{attribute addProperty BoxType "EL3692-0000-0017"}
{attribute addProperty Id "StatusAT %I*Status_888D5AFE1621ValueAT %I*DINT32417"}
{attribute addProperty CRC "1692878231"}
{attribute addProperty SizeInBites "48"}
{attribute addProperty SizeInBytes "6"}
TYPE SAI_Inputs_Channel_64E74597 :
STRUCT
	{attribute addProperty Name "Status"}
	Status AT %I* : Status_888D5AFE;
	{attribute addProperty Name "Value"}
	Value AT %I* : DINT;
END_STRUCT
END_TYPE

(* stored: Version 1.2.0.0, ProductVersion 3.1.4024.9
   DUT SAI_Inputs_Channel_64E74597: Id {479ffae3-a68f-4b74-8fd9-65dcfac1303d} *)
